{attribute 'qualified_only'}
{attribute 'strict'}
TYPE Modbus_map :
(
	enum_member := 0
);
END_TYPE

(* stored: Version 1.1.0.1, ProductVersion 3.1.4024.11
   DUT Modbus_map: Id {8a654f0d-f49b-42d7-a82f-4e34089ae6d6} *)
